ABB RobotStudio station: P2_solucion.rspag

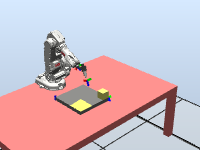
--- station ---
Station P2_paco (saved by RobotStudio 6.6.7701.1025)
Controller Sistema1
  mechanical unit ROB_1: IRB140_6_81_C_03, 6 joints, base frame (1250, 262.2, 836.07) mm, rotated rx 0 ry 0 rz 90 deg
Layout (positions relative to the parent item):
  - Base [part] at (1000, 600, 850) mm
  - Mesa [part]
  - Caja [part]
  - IRB140_6_81_C_03 [mechanism, from Robots\IRB140_6_81_C_G_03.rslib] at (1250, 262.2, 836.07) mm, rotated rx 0 ry 0 rz 90 deg; joint values [0.1248, 0.0655, 0.5598, -2.3067, 0.146, 2.3747] (rad or m)
  - Piramide [part] at (1400, 1000, 900) mm
  - MyTool [mechanism, from Libraries\myTool.rslib] at (1200, 717.02, 1292.35) mm, rotated rx 180 ry 60 rz -90 deg
Attachment: MyTool is attached to IRB140_6_81_C_03 / Link6

--- Backups/Sistema1/RAPID/TASK1/PROGMOD/CalibData.mod ---
MODULE CalibData
	PERS tooldata MyTool:=[TRUE,[[31.792631019,0,229.638935148],[0.945518576,0,0.325568154,0]],[1,[0,0,1],[1,0,0,0],0,0,0]];
    TASK PERS wobjdata placa:=[FALSE,TRUE,"",[[1500,600,850],[0.707106781,0,0,0.707106781]],[[0,0,0],[1,0,0,0]]];
ENDMODULE

--- Backups/Sistema1/RAPID/TASK1/PROGMOD/Module1.mod ---
MODULE Module1
    CONST robtarget P0:=[[500.00004386,500.000013289,49.999987713],[0.190808942,0.000000005,0.981627194,0.000000026],[0,-2,1,0],[9E+09,9E+09,9E+09,9E+09,9E+09,9E+09]];
    CONST robtarget P1:=[[500,-500,50],[0.190808942,0.000000005,0.981627194,0.000000026],[0,-2,1,0],[9E+09,9E+09,9E+09,9E+09,9E+09,9E+09]];



    PROC main()
        cubo;
        cubo_circ;
        piramide;

    ENDPROC

    PROC cubo()

        VAR robtarget esquina1;
        VAR robtarget esquina2;
        VAR robtarget esquina3;
        VAR robtarget esquina4;
        VAR robtarget inicio;


        inicio := Offs(P0,-200,-200,250);
        esquina1 := Offs(P0,2,0,100);
        esquina2 := Offs(P0,2,-103,100);
        esquina3 := Offs(P0,-105,-103,100);
        esquina4 := Offs(P0,-105,0,100);

        MoveL inicio,v300,z10,MyTool\WObj:=placa;
        MoveL esquina1,v300,z10,MyTool\WObj:=placa;
        MoveL esquina2,v300,z10,MyTool\WObj:=placa;
        MoveL esquina3,v300,z10,MyTool\WObj:=placa;
        MoveL esquina4,v300,z10,MyTool\WObj:=placa;
        MoveL esquina1,v300,z10,MyTool\WObj:=placa;
        MoveL inicio,v300,z10,MyTool\WObj:=placa;

    ENDPROC

    PROC cubo_circ()
        VAR robtarget esquina1;
        VAR robtarget esquina2;
        VAR robtarget esquina3;
        VAR robtarget esquina4;
        VAR robtarget inicio;

        inicio := Offs(P0,-200,-200,250);
        esquina1 := Offs(P0,2,0,100);
        esquina2 := Offs(P0,2,-103,100);
        esquina3 := Offs(P0,-105,-103,100);
        esquina4 := Offs(P0,-105,0,100);

        MoveJ inicio,v300,z10,MyTool\WObj:=placa;
        MoveJ esquina1,v300,z10,MyTool\WObj:=placa;
        MoveC esquina2,esquina3,v300,z10,MyTool\WObj:=placa;
        MoveC esquina4,esquina1,v300,z10,MyTool\WObj:=placa;
        MoveJ inicio,v300,z10,MyTool\WObj:=placa;

    ENDPROC


    PROC piramide()

        VAR robtarget esquina1;
        VAR robtarget esquina2;
        VAR robtarget esquina3;
        VAR robtarget esquina4;
        VAR robtarget vertice;
        VAR robtarget verticegir1;
        VAR robtarget verticegir3;
        VAR robtarget esquina1gir;
        VAR robtarget esquina4gir;
        VAR robtarget esquina3gir;
        VAR robtarget esquina2gir;

        VAR robtarget inicio;


        inicio := Offs(P0,-200,-200,250);
        esquina1 := Offs(P0,0,-300,0);
        esquina2 := Offs(P0,0,-500,0);
        esquina3 := Offs(P0,-200,-500,0);
        esquina4 := Offs(P0,-200,-300,000);
        vertice  := Offs(P0,-100,-400,100);

        verticegir1 :=Reltool(vertice,0,0,0, \Rx:=45, \Ry:=45);
        verticegir3 :=Reltool(vertice,0,0,0, \Rx:=15);
        esquina2 :=Reltool(esquina2,0,0,0, \Rx:=15, \Ry:=15);
        esquina1gir :=Reltool(esquina1,0,0,0, \Rx:=15, \RY:=45);
        esquina4gir :=Reltool(esquina4,0,0,0,\Rx:=25,\Rz:=45);
        esquina3gir :=Reltool(esquina3,0,0,0,\Rx:=15,\Rz:=45);
        esquina2gir :=Reltool(esquina2,0,0,0,\Rx:=-15,\Rz:=45);

        MoveJ inicio,v300,z10,MyTool\WObj:=placa;
        MoveL esquina1,v300,z10,MyTool\WObj:=placa;
        MoveL verticegir1,v300,z10,MyTool\WObj:=placa;
        MoveL esquina2,v300,z10,MyTool\WObj:=placa;
        MoveL esquina1gir,v300,z10,MyTool\WObj:=placa;
        MoveL esquina4gir,v300,z10,MyTool\WObj:=placa;
        MoveL verticegir3,v300,z10,MyTool\WObj:=placa;
        MoveL esquina3gir,v300,z10,MyTool\WObj:=placa;
        MoveL esquina2gir,v300,z10,MyTool\WObj:=placa;
        MoveL verticegir1,v300,z10,MyTool\WObj:=placa;
        MoveL esquina3gir,v300,z10,MyTool\WObj:=placa;
        MoveL esquina4gir,v300,z10,MyTool\WObj:=placa;
        MoveJ inicio,v300,z10,MyTool\WObj:=placa;






    ENDPROC



ENDMODULE

--- Backups/Sistema1/RAPID/TASK1/PROGMOD/RsTempModule.mod ---
MODULE RsTempModule
PROC RsTempPath()
ENDPROC
PROC RsTempPath1()
ENDPROC


ENDMODULE

--- Backups/Sistema1/RAPID/TASK1/SYSMOD/LINKEDM.sys ---
%%%
  VERSION:1
  LANGUAGE:ENGLISH
%%%

MODULE LINKEDM (SYSMODULE)

! FOLLOWER
!     Name of electronically linked follower axis used by operator at teach pendent.
      PERS string l_f_axis_name{5}       :=  ["",  "", "", "", ""];

!     Name of the mechanical unit for follower axis.
      PERS string l_f_mecunt_n{5}  :=  ["", "", "", "", ""];

!     Linked follower axis number in the mechanical unit (first axis in mech. unit is number 1).
      PERS num l_f_axis_no{5}      :=  [0,          0,   0,  0,  0];

! MASTER
!     Name of the mechanical unit for linked master axis.
      PERS string l_m_mecunt_n{5} :=  ["", "", "", "", ""];

!     Linked master axis number in the mechanical unit (first axis in mech. unit is number 1).
!     See axis number table in documentation for different master mechanical units.
      PERS num l_m_axis_no{5}     :=  [0,  0,  0,  0,  0];

! POSITION OFFSET
!     The increase of the allowed offset position between the master and follower
!     positions, used when starting AUTO mode. As soon as the offset is decreased
!     the old configurated parameter is used.
!     Example: 3 => the configurated value of allowed offset is increased 3 times.
      PERS num offset_ratio{5}       :=  [10,  10,   10,  10,  10];

! SPEED RATIO
!     Speed_ratio used in AUTO and JOG modes [ very_slow   slow    normal    fast]
!     Value 1 = max allowed manual speed.
      CONST num speed_ratio {20}      := [0.01, 0.01, 0.01, 0.01, 0.01,
                                          0.05, 0.05, 0.05, 0.05, 0.05,
                                          0.20, 0.20, 0.20, 0.20, 0.20,
                                          1.00, 1.00, 1.00, 1.00, 1.00];

! STEP SIZE
!     Displacement position used in JOG mode for each activation of positive or
!     negative movement.                  [very_short    short   normal   long]
!     Unit degees or meter.
      CONST num displacement {20}     := [0.001, 0.001, 0.001, 0.001, 0.001,
                                          0.005, 0.005, 0.005, 0.005, 0.005,
                                          0.020, 0.020, 0.020, 0.020, 0.020,
                                          0.100, 0.100, 0.100, 0.100, 0.100];


!-------------------------------------------------------------
 PROC Linked_m ()
      Linked_m_exe ;
 ENDPROC
ENDMODULE
